{attribute 'qualified_only'}
{attribute 'strict'}
{attribute 'to_string'}
TYPE E_KNXnetIPStateReceivedTelegrams :
(
	eInit 									:= 0,
	eWaitForNextTelegram					:= 1
);
END_TYPE

(* stored: Version 1.1.0.1
   DUT E_KNXnetIPStateReceivedTelegrams: Id {f7a2fadb-f2e3-4198-9191-d589ddf4b706} *)
